FUNCTION_BLOCK FB_ControlMode IMPLEMENTS ITF_ControlModules
VAR_INPUT
    ib_enable      	: BOOL;           // Input to enable the module
    ib_auto        	: BOOL;           // Input to request automatic mode
END_VAR

VAR 
	fault			: ST_ModuleAlarm;  // OPC fault variable
	mode 			: E_Mode;
	requestMode		: E_Mode;
END_VAR

// NOT ENABLE BY PLC
IF NOT ib_enable THEN
	(* If not enabled by PLC , set the module to OFF *)
	mode := E_Mode.OFF;
	M_RaiseFault(description := 'Module disabled', level := E_FaultLevel.DIAGNOSTIC);
// PARENT AUTO REQUEST	
ELSIF ib_auto THEN 
	(* module already in auto *) 
	IF mode = E_Mode.AUTO THEN
		requestMode := E_Mode.AUTO;
		M_RaiseFault(description := 'Controlled by parent system', level := E_FaultLevel.DIAGNOSTIC);
	(* wait to release manual or off mode *)
	ELSIF requestMode = E_Mode.AUTO THEN
		mode := E_Mode.AUTO;
	(* info the parent is requesting auto mode *)
	ELSE
		M_RaiseFault(description := 'Request auto mode from parent system', level := E_FaultLevel.DIAGNOSTIC);
	END_IF
ELSE
	// Manual mode - state is controlled by the HMI input
	mode := requestMode;
	
	// Handle OFF state separately
	IF mode = E_Mode.OFF THEN
		M_RaiseFault(description := 'Module set to OFF by operator', level := E_FaultLevel.DIAGNOSTIC);
	END_IF
END_IF

METHOD M_RaiseFault : BOOL
VAR_INPUT
	description	: STRING;
	level	: E_FaultLevel;
END_VAR
fault.active 		:= TRUE ;
fault.description 	:= description ;
fault.level			:= level;
END_METHOD

METHOD M_ResetFault : BOOL
fault.active 		:= FALSE ;
fault.description 	:= '' ;
fault.level			:= E_FaultLevel.DIAGNOSTIC;
END_METHOD

PROPERTY P_mode : E_Mode;
GET
P_mode := mode;
END_GET
END_PROPERTY

END_FUNCTION_BLOCK

(* stored: Version 1.1.0.1, ProductVersion 3.1.4024.13
   POU FB_ControlMode: Id {aa8165d9-f0a8-4ec7-8af3-232727d4d166}, SpecialFunc None
   Method M_RaiseFault: Id {ade556bc-f5cd-4f29-951a-7f6ee782a652}
   Method M_ResetFault: Id {bb3e0da9-9140-4e16-a72f-5e2c36fc40ff}
   Property P_mode: Id {50587c59-f5d5-444c-82f7-a3afd9aff209}
   Get Get: Id {67a0fd01-3318-4564-8c5f-62654cc15452} *)
